Xinje XDPPro project, PLC1: XD5E-60T10 (software 3.5.3 2018-11-19)

PROGRAM Ladder

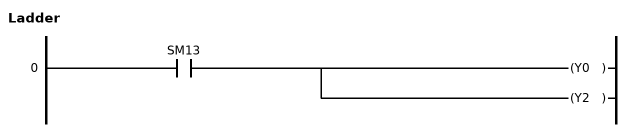
LD     SM13
OUT    Y0
OUT    Y2